# EPICS StreamDevice protocol: streamDevice/shutter.proto
# Sidekick EPICS Shutter protocol file
# Built by examining examples at: https://paulscherrerinstitute.github.io/StreamDevice/protocol.html#gen

Terminator = CR LF;

info {
	ExtraInput = Ignore;
	out "*IDN?";
	in "%39c";
}

# Duration is an unsigned long integer
# Use int64 record type
getDuration {
        out "SHUtter:DURation?";
        in "%u";
    }

setDuration {
        out "SHUtter:DURation %u";
        @init { getDuration; }
    }

getEnable {
        out "SHUtter:ENable?";
        in "%u";
    }

setEnable {
        out "SHUtter:ENable %u";
        @init { getEnable; }
    }

debug {
   ExtraInput = Ignore;
   out "%s";
   in "%39c";
}
